INTERFACE InterfaceEventViewer

METHOD clear : BOOL
VAR_INPUT
END_VAR
END_METHOD

METHOD history_clear : BOOL
VAR_INPUT
END_VAR
END_METHOD

METHOD send_event : BOOL
VAR_INPUT
	event_container : REFERENCE TO EventContainer;
END_VAR
END_METHOD

METHOD show : BOOL
VAR_INPUT
	event_container : REFERENCE TO EventContainer;
END_VAR
END_METHOD

END_INTERFACE

(* stored: Version 1.1.0.1, ProductVersion 3.1.4024.15
   Itf InterfaceEventViewer: Id {f0fe6b76-22c6-4254-b213-56b0ec69b1b9}
   Method clear: Id {1b0ef198-ec53-4b5e-96b9-b8c37507bbe2}
   Method history_clear: Id {2f8fe953-1f5f-4c5e-88cf-74b8b2f74278}
   Method send_event: Id {6944e801-828c-436b-a997-770d62cacb42}
   Method show: Id {8555b326-6a37-41fd-9f1b-f223bb9aeabd} *)
